(* IEC 61131-3 sources: ATCMcontrol_Engineering/src/TargetBase/Libs/ATCM_IEC1131_3/table_30, 4 files *)

(* ---- add_time.st ---- *)
(*[[
    UserURL= "ATCMfile:ADD_TIME.htm"
]]*)

FUNCTION ADD_TIME : TIME
VAR_INPUT
    IN1 : TIME;
    IN2 : TIME;
END_VAR

inline +

END_FUNCTION

(* ---- divtime.st ---- *)
(*[[
    UserURL= "ATCMfile:DIVTIME.htm"
]]*)

FUNCTION DIVTIME : TIME
VAR_INPUT
    IN1 : TIME;
    IN2 : ANY_NUM;
END_VAR

overload TIME(TIME,INT)
inline
{
    %1
    %2
    int_to_dint
    div_dint
}

overload TIME(TIME,DINT)
inline
{
    %1
    %2
    div_dint
}

overload TIME(TIME,REAL)
inline
{
    %1
    dint_to_real
    %2
    div_real
    real_to_dint
}

overload TIME(TIME,LREAL)
inline
{
    %1
    dint_to_lreal
    %2
    div_lreal
    lreal_to_dint
}

END_FUNCTION

(* ---- multime.st ---- *)
(*[[
    UserURL= "ATCMfile:MULTIME.htm"
]]*)

FUNCTION MULTIME : TIME
VAR_INPUT
    IN1 : TIME;
    IN2 : ANY_NUM;
END_VAR

overload TIME(TIME,INT)
inline
{
    %1
    %2
    int_to_dint
    mul_dint
}

overload TIME(TIME,DINT)
inline
{
    %1
    %2
    mul_dint
}

overload TIME(TIME,REAL)
inline
{
    %1
    dint_to_real
    %2
    mul_real
    real_to_dint
}

overload TIME(TIME,LREAL)
inline
{
    %1
    dint_to_lreal
    %2
    mul_lreal
    lreal_to_dint
}

END_FUNCTION

(* ---- sub_time.st ---- *)
(*[[
    UserURL= "ATCMfile:SUB_TIME.htm"
]]*)

FUNCTION SUB_TIME : TIME
VAR_INPUT
    IN1 : TIME;
    IN2 : TIME;
END_VAR

inline -

END_FUNCTION
